# B&R Automation Studio project prac4
Automation Studio 4.5.2.102

## Configuration Config1

CPU 4PP065.0571-P74, AutomationRuntime D4.52, Build 4.1.2, Vc V4.52.0, Safety 1.6

### Task classes (Cpu.sw)
```
Cyclic#1 (cycle 2000 us, tolerance 0 us):
  ncsdcctrl <- ncsdcctrl.prg
Cyclic#4:
  Program <- Program.prg
  Program1 <- Program1.prg
NcDataObjects: acp10etxen <- acp10etxen.dob, gAxis01a <- gAxis01obj.gAxis01a.dob, gAxis01i <- gAxis01obj.gAxis01i.dob, gAxis02a <- gAxis02obj.gAxis02a.dob, gAxis02i <- gAxis02obj.gAxis02i.dob
VcDataObjects: Visu <- Visu.dob
Libraries: Acp10man, Acp10par, NcGlobal, Acp10sdc, AsBrStr, Acp10_MC, brsystem, sys_lib, runtime, Library
```

### Hardware
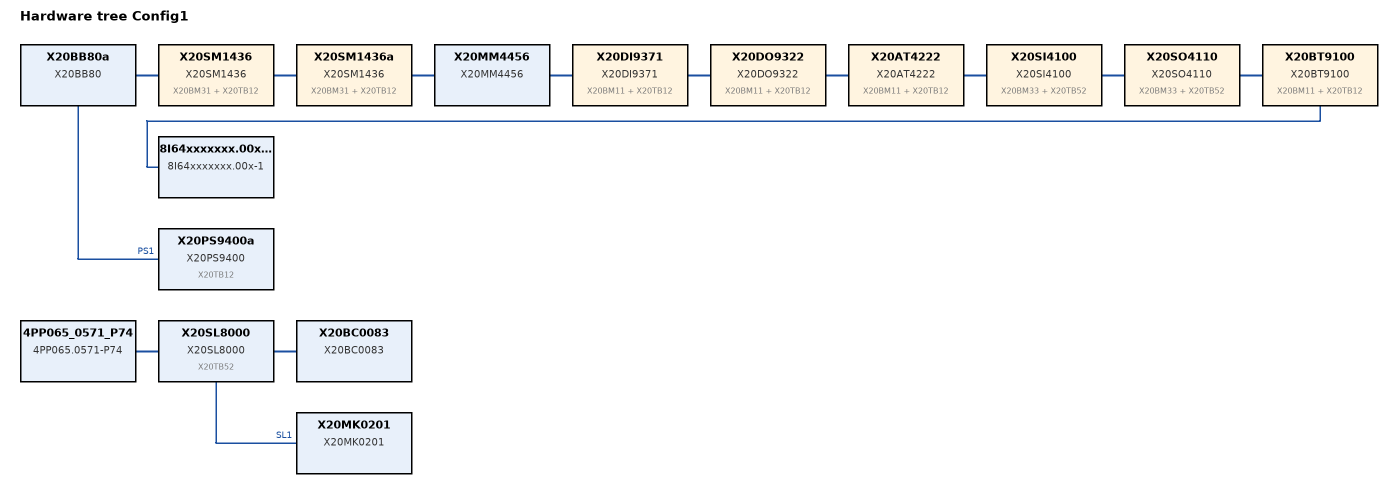
```
4PP065_0571_P74 : 4PP065.0571-P74 v1.1.2.0
  Connector IF5:
    ActivateDevice = 1
    Mode = Manual
    InternetAddress = 10.0.1.4
    SubnetMask = 255.255.255.0
    Vnc1
    VncVcObjectName1 = 
    VncKeyMappingFile1 = 
  ConfigurationID = labBR
  TimerDeviceType = EPLX2X
  TimerDevice = 4PP065_0571_P74.IF4
  TaskClassIdleTime = 2000
  Cyclic1Duration = 2000
  Cyclic1Tolerance = 0
  Cyclic1Output = 1
  VcObjectName = Visu
8I64xxxxxxx.00x-1 : 8I64xxxxxxx.00x-1 v2.1.2.0  [X2X1 -> X20BT9100.X2X1 [Cable Type=X2XCable, Length=10, Version=1.0.0.2]]
  packedETAD = packed
  packedCMDD = packed
X20AT4222 : X20AT4222 v1.2.3.0  [SS1 -> X20TB12e.SS; SL -> X20BM11b.SL1]
X20BB80a : X20BB80 v1.0.2.0
X20BC0083 : X20BC0083 v2.9.0.0  [PLK1 -> X20SL8000.PLK2 [Cable Type=PowerlinkCable, Length=10, Version=1.0.0.2]; SL -> X20BB80a.SL1]
X20BM11 : X20BM11 v1.0.0.1  [X2X1 -> X20MM4456.X2X2]
X20BM11a : X20BM11 v1.0.0.1  [X2X1 -> X20BM11.X2X2]
X20BM11b : X20BM11 v1.0.0.1  [X2X1 -> X20BM11a.X2X2]
X20BM11c : X20BM11 v1.0.0.1  [X2X1 -> X20BM33a.X2X2]
X20BM31 : X20BM31 v1.0.0.1  [X2X1 -> X20BB80a.IF1]
X20BM31a : X20BM31 v1.0.0.1  [X2X1 -> X20BM31.X2X2]
X20BM33 : X20BM33 v1.0.0.4  [X2X1 -> X20BM11b.X2X2]
X20BM33a : X20BM33 v1.0.0.4  [X2X1 -> X20BM33.X2X2]
X20BT9100 : X20BT9100 v1.0.3.0  [SS1 -> X20TB12f.SS; SL -> X20BM11c.SL1]
X20DI9371 : X20DI9371 v1.0.2.0  [SS1 -> X20TB12c.SS; SL -> X20BM11.SL1]
X20DO9322 : X20DO9322 v1.0.3.0  [SS1 -> X20TB12d.SS; SL -> X20BM11a.SL1]
X20MK0201 : X20MK0201 v1.0.0.0  [SL -> X20SL8000.SL1]
X20MM4456 : X20MM4456 v1.1.5.0  [X2X1 -> X20BM31a.X2X2]
X20PS9400a : X20PS9400 v1.0.2.4  [SS1 -> X20TB12a.SS; PS -> X20BB80a.PS1]
X20SI4100 : X20SI4100 v1.10.1.1  [SS1 -> X20TB52a.SS; SL -> X20BM33.SL1]
X20SL8000 : X20SL8000 v1.6.5.1  [PLK1 -> 4PP065_0571_P74.IF4 [Cable Type=PowerlinkCable, Length=10, Version=1.0.0.2]; PLK2 -> X20BC0083.PLK1 [Cable Type=PowerlinkCable, Length=10, Version=1.0.0.2]; SS1 -> X20TB52.SS]
  SafeProject = SafeLOGIC-1
X20SM1436 : X20SM1436 v1.4.2.1  [SS1 -> X20TB12.SS; SL -> X20BM31.SL1]
X20SM1436a : X20SM1436 v1.4.2.1  [SS1 -> X20TB12b.SS; SL -> X20BM31a.SL1]
X20SO4110 : X20SO4110 v1.10.1.1  [SS1 -> X20TB52b.SS; SL -> X20BM33a.SL1]
  SafeModuleID = 3
X20TB12 : X20TB12 v1.0.0.0
X20TB12a : X20TB12 v1.0.0.0
X20TB12b : X20TB12 v1.0.0.0
X20TB12c : X20TB12 v1.0.0.0
X20TB12d : X20TB12 v1.0.0.0
X20TB12e : X20TB12 v1.0.0.0
X20TB12f : X20TB12 v1.0.0.0
X20TB52 : X20TB52 v1.0.0.1
X20TB52a : X20TB52 v1.0.0.1
X20TB52b : X20TB52 v1.0.0.1
```

### IoMap.iom - 4PP065_0571_P74/IoMap.iom
```iecst
VAR_CONFIG
	Cyclic#1.gAxis02_DrvIf.iLifeCnt AT %IB."8I64xxxxxxx.00x-1".SDC_LifeCnt;
	Cyclic#1.gAxis02_DrvIf.iDrvOK AT %IX."8I64xxxxxxx.00x-1".ETAD_Input_Bool_02;
	Cyclic#1.gAxis02_DrvIf.oSetTime AT %QW."8I64xxxxxxx.00x-1".SDC_SetTime;
	::Program:speed AT %QW."8I64xxxxxxx.00x-1".LFRD_Output;
	Cyclic#1.gAxis02_DiDoIf.iLifeCntDriveReady AT %IB."8I64xxxxxxx.00x-1".SDC_LifeCnt;
	Cyclic#1.gAxis02_DiDoIf.iLifeCntDriveEnable AT %IB."8I64xxxxxxx.00x-1".SDC_LifeCnt;
	Cyclic#1.gAxis02_DiDoIf.oDriveEnable AT %QX."8I64xxxxxxx.00x-1".CMDD_Output_Bool_00;
	Cyclic#1.gAxis02_ModuleOk AT %QX."8I64xxxxxxx.00x-1".CMDD_Output_Bool_01;
	Cyclic#1.gAxis02_ModuleOk AT %QX."8I64xxxxxxx.00x-1".CMDD_Output_Bool_02;
	Cyclic#1.gAxis02_ModuleOk AT %IX."8I64xxxxxxx.00x-1".ModuleOk;
	Cyclic#1.gAxis02_DiDoIf.oDriveEnable AT %QX."8I64xxxxxxx.00x-1".CMDD_Output_Bool_03;
	Cyclic#1.gAxis02_DiDoIf.iDriveReady AT %IX."8I64xxxxxxx.00x-1".ETAD_Input_Bool_02;
	EVIRD.STATE AT %IW."8I64xxxxxxx.00x-1".ETAD_Input;
	::EVIRD.COM AT %QW."8I64xxxxxxx.00x-1".CMDD_Output;
	::led1 AT %QX."X20DO9322".DigitalOutput02;
	::led2 AT %QX."X20DO9322".DigitalOutput03;
	::led3 AT %QX."X20DO9322".DigitalOutput04;
	::led4 AT %QX."X20DO9322".DigitalOutput05;
	::EVIRD.real_speed AT %IW."8I64xxxxxxx.00x-1".RFRD_Input;
END_VAR
```

## Logical view

Binary libraries used (declarations not repeated): astime, operator, runtime, AsIecCon, Acp10man, Acp10par, NcGlobal, Acp10sdc, AsBrStr, brsystem, sys_lib, Acp10_MC, Library


### Program Logical/Program (ANSIC)

#### Main.c
```c
#include <bur/plctypes.h>

#ifdef _DEFAULT_INCLUDES
	#include <AsDefault.h>
#endif

void _INIT ProgramInit(void)
{
	speed = 500;
	EVIRD.ENABLE=1;
}

void _CYCLIC ProgramCyclic(void)
{

	DRIVE(&EVIRD);
}

void _EXIT ProgramExit(void)
{

}
```

### Program Logical/Program1 (ANSIC)

#### Variables.var
```iecst
VAR
	LED : ARRAY[0..3] OF BOOL;
	ACTIV : INT := 0;
	i : INT := 0;
END_VAR
```

#### Main.c
```c
#include <bur/plctypes.h>

#ifdef _DEFAULT_INCLUDES
	#include <AsDefault.h>
#endif

void _INIT ProgramInit(void)
{
	i = 0;
}

void _CYCLIC ProgramCyclic(void)
{
	led1 = LED[0];
	led2 = LED[1];
	led3 = LED[2];
	led4 = LED[3];
	if(active_deactive_taming==1){
		led1=!led1;
		if(i%5==0){led1=!led1;}
		if(i%10==0){led2=!led2;}
		if(i%20==0){led3=!led3;}
		if(i%30==0){led4=!led4;}
		i++;
	}
}

void _EXIT ProgramExit(void)
{

}
```

- Visualisation Logical/Visu (not shown)

### Global.var - Global variables
```iecst
VAR
	gAxis02_HW : SdcHwCfg_typ := (0);
	gAxis01_HW : SdcHwCfg_typ := (0);
	gAxis02_DrvIf : SdcDrvIf16_typ := (0);
	gAxis01_DrvIf : SdcDrvIf16_typ := (0);
	gAxis02_DiDoIf : SdcDiDoIf_typ := (0);
	gAxis01_DiDoIf : SdcDiDoIf_typ := (0);
	EVIRD : DRIVE;
	led4 : BOOL;
	led3 : BOOL;
	led2 : BOOL;
	led1 : BOOL;
	gAxis02_ModuleOk : BOOL := 0;
	gAxis01_ModuleOk : BOOL := 0;
	gAxis02 : ACP10AXIS_typ;
	gAxis01 : ACP10AXIS_typ;
	i : INT := 0;
	active_deactive_taming : BOOL;
END_VAR
```

Listed in the project but not available here: Logical/Global.typ, Logical/acp10etxen, Logical/ncsdcctrl, Logical/gAxis01obj, Logical/gAxis02obj
